// TIA Portal V21 export
FUNCTION "GestSensore" : Void   // FC9, LAD
{ S7_Optimized_Access := 'TRUE' }
// stored: SetENOAutomatically false
   VAR_INPUT
      K_Sensore : Int;
      K_TipoSensore : Int;
      K_Zona : Int;
   END_VAR
BEGIN
END_FUNCTION
